// Mitsubishi GX Works2 project: LRI - Exercìcio 6   PLC: Q03UDV
// HelloWorld

PROGRAM MAIN
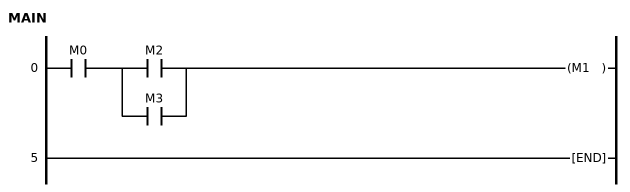
0     LD      M0
      LD      M2
      OR      M3
      ANB
      OUT     M1
5     END
END_PROGRAM
